// TwinCAT 3 PLC project LAMPKB
// ProgramVersion: 3.1.4023.0
// libraries:
//   LCLS General, * (SLAC)
//   lcls-twincat-motion, * (SLAC)
//   Tc2_MC2, * (Beckhoff Automation GmbH)
//   Tc2_Standard, * (Beckhoff Automation GmbH)
//   Tc2_System, * (Beckhoff Automation GmbH)
//   Tc3_Module, * (Beckhoff Automation GmbH)
// project tree:
//   / PlcTask.TcTTO
//   POUs/ FB_MotionStageStats.TcPOU, FB_PAT.TcPOU, MAIN.TcPOU
// real-time tasks:
//   TASK PlcTask: cycle T#10ms, priority 20, ADS port 350
// motion (NC):
//   TASK NC-Task 1 SAF: cycle T#2ms, priority 4, ADS port 501
//   TASK NC-Task 1 SVB: cycle T#10ms, priority 8, ADS port 511
//   AXIS MR2K4 X (id 1)
//     Dynamic: AccelerationMaximum=100, DecelerationMaximum=100, Acceleration=100, Deceleration=100, DelayTime=0.008
//     Velo: Maximum=20
//     OtherSettings: AllowMotionCmdToSlave=true
//     encoder EncType=29
//       EncPara: ScaleFactorNumerator=5e-06, Offset=-30.6825, MaxCount=#xffffffff, ReferenceSystem=1
//         Inc: RefSoftSyncMask=#x0000ffff
//     drive DrvType=24
//       DrvPara: Inverse=true
//         Analog: VeloReferenz=20, ScaleFactorActTorque=0.1
//         TimeComp: TaskDelayCycles=1
//     controller CtrType=1
//       CtrPara: PriorControlFactor=1
//         PosDiffControl: Range=0.1
//         PID: DeadBandPosition=0.001
//         Observer: BandWidth=20
//   AXIS MR2K4 Y (id 2)
//     Dynamic: AccelerationMaximum=10, DecelerationMaximum=10, Acceleration=10, Deceleration=10, Jerk=15, DelayTime=0.008
//     Velo: Maximum=1.25
//     OtherSettings: AllowMotionCmdToSlave=true
//     encoder EncType=29
//       EncPara: ScaleFactorNumerator=5e-06, Offset=-30.18, MaxCount=#xffffffff
//         Inc: RefSoftSyncMask=#x0000ffff
//     drive DrvType=24
//       DrvPara: Inverse=true
//         Analog: VeloReferenz=1.25, ScaleFactorActTorque=0.1
//         TimeComp: TaskDelayCycles=1
//     controller CtrType=1
//       CtrPara: PriorControlFactor=1
//         PosDiffControl: Range=0.1
//         Observer: BandWidth=20
//   AXIS MR2K4 rY (id 3)
//     General: UnitName=urad
//     Dynamic: AccelerationMaximum=400, DecelerationMaximum=400, Acceleration=400, Deceleration=400, Jerk=1200, DelayTime=0.008
//     Velo: Maximum=166.67
//     OtherSettings: AllowMotionCmdToSlave=true
//     encoder EncType=29
//       EncPara: ScaleFactorNumerator=0.005348, Offset=-194502.025, MaxCount=#xffffffff
//         Inc: RefSoftSyncMask=#x0000ffff
//     drive DrvType=24
//       Analog: VeloReferenz=166.67, ScaleFactorActTorque=0.1
//       TimeComp: TaskDelayCycles=1
//     controller CtrType=1
//       CtrPara: PriorControlFactor=1
//         PosDiffControl: Range=40
//         Observer: BandWidth=20
//   AXIS MR3K4 X (id 4)
//     Dynamic: AccelerationMaximum=100, DecelerationMaximum=100, Acceleration=100, Deceleration=100, DelayTime=0.008
//     Velo: Maximum=20
//     OtherSettings: AllowMotionCmdToSlave=true
//     encoder EncType=29
//       EncPara: ScaleFactorNumerator=5e-06, Offset=-31.1, MaxCount=#xffffffff
//         Inc: RefSoftSyncMask=#x0000ffff
//     drive DrvType=24
//       DrvPara: Inverse=true
//         Analog: VeloReferenz=20, ScaleFactorActTorque=0.1
//         TimeComp: TaskDelayCycles=1
//     controller CtrType=1
//       CtrPara: PriorControlFactor=1
//         PosDiffControl: Range=0.1
//         Observer: BandWidth=20
//   AXIS MR3K4 Y (id 5)
//     Dynamic: AccelerationMaximum=10, DecelerationMaximum=10, Acceleration=10, Deceleration=10, Jerk=15, DelayTime=0.008
//     Velo: Maximum=1.25
//     OtherSettings: AllowMotionCmdToSlave=true
//     encoder EncType=29
//       EncPara: ScaleFactorNumerator=5e-06, Offset=-29.68, MaxCount=#xffffffff
//         Inc: RefSoftSyncMask=#x0000ffff
//     drive DrvType=24
//       DrvPara: Inverse=true
//         Analog: VeloReferenz=1.25, ScaleFactorActTorque=0.1
//         TimeComp: TaskDelayCycles=1
//     controller CtrType=1
//       CtrPara: PriorControlFactor=1
//         PosDiffControl: Range=0.1
//         Observer: BandWidth=20
//   AXIS MR3K4 rX (id 6)
//     General: UnitName=urad
//     Dynamic: AccelerationMaximum=300, DecelerationMaximum=300, Acceleration=300, Deceleration=300, Jerk=900, DelayTime=0.008
//     Velo: Maximum=140.84
//     OtherSettings: AllowMotionCmdToSlave=true
//     encoder EncType=29
//       EncPara: ScaleFactorNumerator=0.002577, Offset=-136547, MaxCount=#xffffffff
//         Inc: RefSoftSyncMask=#x0000ffff
//     drive DrvType=24
//       Analog: VeloReferenz=140.84, ScaleFactorActTorque=0.1
//       TimeComp: TaskDelayCycles=1
//     controller CtrType=1
//       CtrPara: PriorControlFactor=1
//         PosDiffControl: Range=10
//         Observer: BandWidth=20
//   AXIS MR2K4 BEND US (id 14)
//     Dynamic: AccelerationMaximum=0.6, DecelerationMaximum=0.6, Acceleration=0.6, Deceleration=0.6, Jerk=1.2, DelayTime=0.008
//     Velo: Maximum=0.4
//     OtherSettings: AllowMotionCmdToSlave=true
//     encoder EncType=29
//       EncPara: ScaleFactorNumerator=1e-06, MaxCount=#xffffffff
//         SoftEndMinControl: Enable=true, Range=5
//         Inc: RefSoftSyncMask=#x0000ffff
//     drive DrvType=24
//       DrvPara: Inverse=true
//         Analog: VeloReferenz=0.4, ScaleFactorActTorque=0.1
//         TimeComp: TaskDelayCycles=1
//     controller CtrType=1
//       CtrPara: PriorControlFactor=1
//         PosDiffControl: Range=0.2
//         Observer: BandWidth=20
//   AXIS MR2K4 BEND DS (id 15)
//     Dynamic: AccelerationMaximum=0.6, DecelerationMaximum=0.6, Acceleration=0.6, Deceleration=0.6, Jerk=1.2, DelayTime=0.008
//     Velo: Maximum=0.1
//     OtherSettings: AllowMotionCmdToSlave=true
//     encoder EncType=29
//       EncPara: ScaleFactorNumerator=1e-06, MaxCount=#xffffffff
//         SoftEndMinControl: Enable=true, Range=5
//         Inc: RefSoftSyncMask=#x0000ffff
//     drive DrvType=24
//       DrvPara: Inverse=true
//         Analog: VeloReferenz=0.4, ScaleFactorActTorque=0.1
//         TimeComp: TaskDelayCycles=1
//     controller CtrType=1
//       CtrPara: PriorControlFactor=1
//         PosDiffControl: Range=0.2
//         Observer: BandWidth=20
//   AXIS MR3K4 BEND US (id 16)
//     Dynamic: AccelerationMaximum=0.6, DecelerationMaximum=0.6, Acceleration=0.6, Deceleration=0.6, Jerk=1.2, DelayTime=0.008
//     Velo: Maximum=0.1
//     OtherSettings: AllowMotionCmdToSlave=true
//     encoder EncType=29
//       EncPara: ScaleFactorNumerator=1e-06, MaxCount=#xffffffff
//         SoftEndMinControl: Enable=true, Range=6.25
//         Inc: RefSoftSyncMask=#x0000ffff
//     drive DrvType=24
//       DrvPara: Inverse=true
//         Analog: VeloReferenz=0.4, ScaleFactorActTorque=0.1
//         TimeComp: TaskDelayCycles=1
//     controller CtrType=1
//       CtrPara: PriorControlFactor=1
//         PosDiffControl: Range=0.2
//         Observer: BandWidth=20
//   AXIS MR3K4 BEND DS (id 17)
//     Dynamic: AccelerationMaximum=0.6, DecelerationMaximum=0.6, Acceleration=0.6, Deceleration=0.6, Jerk=1.2, DelayTime=0.008
//     Velo: Maximum=0.1
//     OtherSettings: AllowMotionCmdToSlave=true
//     encoder EncType=29
//       EncPara: ScaleFactorNumerator=1e-06, MaxCount=#xffffffff
//         SoftEndMinControl: Enable=true, Range=5.5
//         Inc: RefSoftSyncMask=#x0000ffff
//     drive DrvType=24
//       DrvPara: Inverse=true
//         Analog: VeloReferenz=0.4, ScaleFactorActTorque=0.1
//         TimeComp: TaskDelayCycles=1
//     controller CtrType=1
//       CtrPara: PriorControlFactor=1
//         PosDiffControl: Range=0.2
//         Observer: BandWidth=20
// I/O:
//   DEVICE Device 2 (EtherCAT), AmsNetId 192.168.5.67.3.1
//     Term 1 (EK1100) [EK1100 EtherCAT Coupler (2A E-Bus)]
//       Term 2 (EL5042) [EL5042 2Ch. BiSS-C Encoder]
//       Term 3 (EL5042) [EL5042 2Ch. BiSS-C Encoder]
//       Term 4 (EL5042) [EL5042 2Ch. BiSS-C Encoder]
//       MR2K4 X
//       MR2K4 Y
//       MR2K4 rY
//       MR3K4 X [EL7041-0052 1Ch. Stepper motor output stage (50V, 5A)]
//       MR3K4 Y
//       MR3K4 rX
//       Term 11 (EL9410) [EL9410 E-Bus Power Supplier  (Diagnostics)]
//       Term 12 (EL5042) [EL5042 2Ch. BiSS-C Encoder]
//       Term 13 (EL5042) [EL5042 2Ch. BiSS-C Encoder]
//       MR2K4 BEND US [EL7041 1Ch. Stepper motor output stage (50V, 5A)]
//       MR2K4 BEND DS [EL7041 1Ch. Stepper motor output stage (50V, 5A)]
//       MR3K4 BEND US
//       MR3K4 BEND DS
//       STO (EL1004) [EL1004 4Ch. Dig. Input 24V, 3ms]
//       Term 19 (EL9011) [EL9011 End Terminal]
// variable links:
//   (this object) <-> Device 2 (EtherCAT)/Term 1 (EK1100)/MR2K4 X
//     Drive/Inputs/In/nState1 @bit 3 <-> STM Status/Status/Error
//     Drive/Inputs/In/nState1 @bit 5 <-> STM Status/Status/Moving negative
//     Drive/Inputs/In/nState1 @bit 4 <-> STM Status/Status/Moving positive
//     Drive/Inputs/In/nState1 @bit 1 <-> STM Status/Status/Ready
//     Drive/Inputs/In/nState1 <-> STM Status/Status/Ready to enable
//     Drive/Inputs/In/nState1 @bit 6 <-> STM Status/Status/Torque reduced
//     Drive/Inputs/In/nState1 @bit 2 <-> STM Status/Status/Warning
//     Drive/Inputs/In/nState2 @bit 3 <-> STM Status/Status/Digital input 1
//     Drive/Inputs/In/nState2 @bit 4 <-> STM Status/Status/Digital input 2
//     Drive/Inputs/In/nState2 @bit 5 <-> STM Status/Status/Sync error
//     Drive/Inputs/In/nState2 @bit 7 <-> STM Status/Status/TxPDO Toggle
//     Drive/Inputs/In/nState4 @bit 1 <-> WcState/InputToggle
//     Drive/Inputs/In/nState4 <-> WcState/WcState
//     Drive/Outputs/Out/nCtrl1 <-> STM Control/Control/Enable
//     Drive/Outputs/Out/nCtrl1 @bit 2 <-> STM Control/Control/Reduce torque
//     Drive/Outputs/Out/nCtrl1 @bit 1 <-> STM Control/Control/Reset
//     Drive/Outputs/Out/nDataOut2[0] <-> STM Velocity/Velocity
//   (this object) <-> Device 2 (EtherCAT)/Term 1 (EK1100)/Term 2 (EL5042)
//     Enc/Inputs/In/nComState @bit 1 <-> WcState/InputToggle
//     Enc/Inputs/In/nComState <-> WcState/WcState
//     Enc/Inputs/In/nDataIn1 <-> FB Inputs Channel 1/Position
//     Enc/Inputs/In/nDataIn1 <-> FB Inputs Channel 2/Position
//     Enc/Inputs/In/nState1 @bit 12 <-> FB Inputs Channel 1/Status/Diag
//     Enc/Inputs/In/nState1 @bit 12 <-> FB Inputs Channel 2/Status/Diag
//     Enc/Inputs/In/nState1 @bit 1 <-> FB Inputs Channel 1/Status/Error
//     Enc/Inputs/In/nState1 @bit 1 <-> FB Inputs Channel 2/Status/Error
//     Enc/Inputs/In/nState1 @bit 14 <-> FB Inputs Channel 1/Status/Input cycle counter
//     Enc/Inputs/In/nState1 @bit 14 <-> FB Inputs Channel 2/Status/Input cycle counter
//     Enc/Inputs/In/nState1 @bit 2 <-> FB Inputs Channel 1/Status/Ready
//     Enc/Inputs/In/nState1 @bit 2 <-> FB Inputs Channel 2/Status/Ready
//     Enc/Inputs/In/nState1 @bit 13 <-> FB Inputs Channel 1/Status/TxPDO State
//     Enc/Inputs/In/nState1 @bit 13 <-> FB Inputs Channel 2/Status/TxPDO State
//     Enc/Inputs/In/nState1 <-> FB Inputs Channel 1/Status/Warning
//     Enc/Inputs/In/nState1 <-> FB Inputs Channel 2/Status/Warning
//   (this object) <-> Device 2 (EtherCAT)/Term 1 (EK1100)/MR2K4 Y
//     Drive/Inputs/In/nState1 @bit 3 <-> STM Status/Status/Error
//     Drive/Inputs/In/nState1 @bit 5 <-> STM Status/Status/Moving negative
//     Drive/Inputs/In/nState1 @bit 4 <-> STM Status/Status/Moving positive
//     Drive/Inputs/In/nState1 @bit 1 <-> STM Status/Status/Ready
//     Drive/Inputs/In/nState1 <-> STM Status/Status/Ready to enable
//     Drive/Inputs/In/nState1 @bit 6 <-> STM Status/Status/Torque reduced
//     Drive/Inputs/In/nState1 @bit 2 <-> STM Status/Status/Warning
//     Drive/Inputs/In/nState2 @bit 3 <-> STM Status/Status/Digital input 1
//     Drive/Inputs/In/nState2 @bit 4 <-> STM Status/Status/Digital input 2
//     Drive/Inputs/In/nState2 @bit 5 <-> STM Status/Status/Sync error
//     Drive/Inputs/In/nState2 @bit 7 <-> STM Status/Status/TxPDO Toggle
//     Drive/Inputs/In/nState4 @bit 1 <-> WcState/InputToggle
//     Drive/Inputs/In/nState4 <-> WcState/WcState
//     Drive/Outputs/Out/nCtrl1 <-> STM Control/Control/Enable
//     Drive/Outputs/Out/nCtrl1 @bit 2 <-> STM Control/Control/Reduce torque
//     Drive/Outputs/Out/nCtrl1 @bit 1 <-> STM Control/Control/Reset
//     Drive/Outputs/Out/nDataOut2[0] <-> STM Velocity/Velocity
//   (this object) <-> Device 2 (EtherCAT)/Term 1 (EK1100)/MR2K4 rY
//     Drive/Inputs/In/nState1 @bit 3 <-> STM Status/Status/Error
//     Drive/Inputs/In/nState1 @bit 5 <-> STM Status/Status/Moving negative
//     Drive/Inputs/In/nState1 @bit 4 <-> STM Status/Status/Moving positive
//     Drive/Inputs/In/nState1 @bit 1 <-> STM Status/Status/Ready
//     Drive/Inputs/In/nState1 <-> STM Status/Status/Ready to enable
//     Drive/Inputs/In/nState1 @bit 6 <-> STM Status/Status/Torque reduced
//     Drive/Inputs/In/nState1 @bit 2 <-> STM Status/Status/Warning
//     Drive/Inputs/In/nState2 @bit 3 <-> STM Status/Status/Digital input 1
//     Drive/Inputs/In/nState2 @bit 4 <-> STM Status/Status/Digital input 2
//     Drive/Inputs/In/nState2 @bit 5 <-> STM Status/Status/Sync error
//     Drive/Inputs/In/nState2 @bit 7 <-> STM Status/Status/TxPDO Toggle
//     Drive/Inputs/In/nState4 @bit 1 <-> WcState/InputToggle
//     Drive/Inputs/In/nState4 <-> WcState/WcState
//     Drive/Outputs/Out/nCtrl1 <-> STM Control/Control/Enable
//     Drive/Outputs/Out/nCtrl1 @bit 2 <-> STM Control/Control/Reduce torque
//     Drive/Outputs/Out/nCtrl1 @bit 1 <-> STM Control/Control/Reset
//     Drive/Outputs/Out/nDataOut2[0] <-> STM Velocity/Velocity
//   (this object) <-> Device 2 (EtherCAT)/Term 1 (EK1100)/Term 3 (EL5042)
//     Enc/Inputs/In/nComState @bit 1 <-> WcState/InputToggle
//     Enc/Inputs/In/nComState <-> WcState/WcState
//     Enc/Inputs/In/nDataIn1 <-> FB Inputs Channel 1/Position
//     Enc/Inputs/In/nDataIn1 <-> FB Inputs Channel 2/Position
//     Enc/Inputs/In/nState1 @bit 12 <-> FB Inputs Channel 1/Status/Diag
//     Enc/Inputs/In/nState1 @bit 12 <-> FB Inputs Channel 2/Status/Diag
//     Enc/Inputs/In/nState1 @bit 1 <-> FB Inputs Channel 1/Status/Error
//     Enc/Inputs/In/nState1 @bit 1 <-> FB Inputs Channel 2/Status/Error
//     Enc/Inputs/In/nState1 @bit 14 <-> FB Inputs Channel 1/Status/Input cycle counter
//     Enc/Inputs/In/nState1 @bit 14 <-> FB Inputs Channel 2/Status/Input cycle counter
//     Enc/Inputs/In/nState1 @bit 2 <-> FB Inputs Channel 1/Status/Ready
//     Enc/Inputs/In/nState1 @bit 2 <-> FB Inputs Channel 2/Status/Ready
//     Enc/Inputs/In/nState1 @bit 13 <-> FB Inputs Channel 1/Status/TxPDO State
//     Enc/Inputs/In/nState1 @bit 13 <-> FB Inputs Channel 2/Status/TxPDO State
//     Enc/Inputs/In/nState1 <-> FB Inputs Channel 1/Status/Warning
//     Enc/Inputs/In/nState1 <-> FB Inputs Channel 2/Status/Warning
//   (this object) <-> Device 2 (EtherCAT)/Term 1 (EK1100)/MR3K4 X
//     Drive/Inputs/In/nState1 @bit 3 <-> STM Status/Status/Error
//     Drive/Inputs/In/nState1 @bit 5 <-> STM Status/Status/Moving negative
//     Drive/Inputs/In/nState1 @bit 4 <-> STM Status/Status/Moving positive
//     Drive/Inputs/In/nState1 @bit 1 <-> STM Status/Status/Ready
//     Drive/Inputs/In/nState1 <-> STM Status/Status/Ready to enable
//     Drive/Inputs/In/nState1 @bit 6 <-> STM Status/Status/Torque reduced
//     Drive/Inputs/In/nState1 @bit 2 <-> STM Status/Status/Warning
//     Drive/Inputs/In/nState2 @bit 3 <-> STM Status/Status/Digital input 1
//     Drive/Inputs/In/nState2 @bit 4 <-> STM Status/Status/Digital input 2
//     Drive/Inputs/In/nState2 @bit 5 <-> STM Status/Status/Sync error
//     Drive/Inputs/In/nState2 @bit 7 <-> STM Status/Status/TxPDO Toggle
//     Drive/Inputs/In/nState4 @bit 1 <-> WcState/InputToggle
//     Drive/Inputs/In/nState4 <-> WcState/WcState
//     Drive/Outputs/Out/nCtrl1 <-> STM Control/Control/Enable
//     Drive/Outputs/Out/nCtrl1 @bit 2 <-> STM Control/Control/Reduce torque
//     Drive/Outputs/Out/nCtrl1 @bit 1 <-> STM Control/Control/Reset
//     Drive/Outputs/Out/nDataOut2[0] <-> STM Velocity/Velocity
//   (this object) <-> Device 2 (EtherCAT)/Term 1 (EK1100)/MR3K4 Y
//     Drive/Inputs/In/nState1 @bit 3 <-> STM Status/Status/Error
//     Drive/Inputs/In/nState1 @bit 5 <-> STM Status/Status/Moving negative
//     Drive/Inputs/In/nState1 @bit 4 <-> STM Status/Status/Moving positive
//     Drive/Inputs/In/nState1 @bit 1 <-> STM Status/Status/Ready
//     Drive/Inputs/In/nState1 <-> STM Status/Status/Ready to enable
//     Drive/Inputs/In/nState1 @bit 6 <-> STM Status/Status/Torque reduced
//     Drive/Inputs/In/nState1 @bit 2 <-> STM Status/Status/Warning
//     Drive/Inputs/In/nState2 @bit 3 <-> STM Status/Status/Digital input 1
//     Drive/Inputs/In/nState2 @bit 4 <-> STM Status/Status/Digital input 2
//     Drive/Inputs/In/nState2 @bit 5 <-> STM Status/Status/Sync error
//     Drive/Inputs/In/nState2 @bit 7 <-> STM Status/Status/TxPDO Toggle
//     Drive/Inputs/In/nState4 @bit 1 <-> WcState/InputToggle
//     Drive/Inputs/In/nState4 <-> WcState/WcState
//     Drive/Outputs/Out/nCtrl1 <-> STM Control/Control/Enable
//     Drive/Outputs/Out/nCtrl1 @bit 2 <-> STM Control/Control/Reduce torque
//     Drive/Outputs/Out/nCtrl1 @bit 1 <-> STM Control/Control/Reset
//     Drive/Outputs/Out/nDataOut2[0] <-> STM Velocity/Velocity
//   (this object) <-> Device 2 (EtherCAT)/Term 1 (EK1100)/Term 4 (EL5042)
//     Enc/Inputs/In/nComState @bit 1 <-> WcState/InputToggle
//     Enc/Inputs/In/nComState <-> WcState/WcState
//     Enc/Inputs/In/nDataIn1 <-> FB Inputs Channel 1/Position
//     Enc/Inputs/In/nDataIn1 <-> FB Inputs Channel 2/Position
//     Enc/Inputs/In/nState1 @bit 12 <-> FB Inputs Channel 1/Status/Diag
//     Enc/Inputs/In/nState1 @bit 12 <-> FB Inputs Channel 2/Status/Diag
//     Enc/Inputs/In/nState1 @bit 1 <-> FB Inputs Channel 1/Status/Error
//     Enc/Inputs/In/nState1 @bit 1 <-> FB Inputs Channel 2/Status/Error
//     Enc/Inputs/In/nState1 @bit 14 <-> FB Inputs Channel 1/Status/Input cycle counter
//     Enc/Inputs/In/nState1 @bit 14 <-> FB Inputs Channel 2/Status/Input cycle counter
//     Enc/Inputs/In/nState1 @bit 2 <-> FB Inputs Channel 1/Status/Ready
//     Enc/Inputs/In/nState1 @bit 2 <-> FB Inputs Channel 2/Status/Ready
//     Enc/Inputs/In/nState1 @bit 13 <-> FB Inputs Channel 1/Status/TxPDO State
//     Enc/Inputs/In/nState1 @bit 13 <-> FB Inputs Channel 2/Status/TxPDO State
//     Enc/Inputs/In/nState1 <-> FB Inputs Channel 1/Status/Warning
//     Enc/Inputs/In/nState1 <-> FB Inputs Channel 2/Status/Warning
//   (this object) <-> Device 2 (EtherCAT)/Term 1 (EK1100)/MR3K4 rX
//     Drive/Inputs/In/nState1 @bit 3 <-> STM Status/Status/Error
//     Drive/Inputs/In/nState1 @bit 5 <-> STM Status/Status/Moving negative
//     Drive/Inputs/In/nState1 @bit 4 <-> STM Status/Status/Moving positive
//     Drive/Inputs/In/nState1 @bit 1 <-> STM Status/Status/Ready
//     Drive/Inputs/In/nState1 <-> STM Status/Status/Ready to enable
//     Drive/Inputs/In/nState1 @bit 6 <-> STM Status/Status/Torque reduced
//     Drive/Inputs/In/nState1 @bit 2 <-> STM Status/Status/Warning
//     Drive/Inputs/In/nState2 @bit 3 <-> STM Status/Status/Digital input 1
//     Drive/Inputs/In/nState2 @bit 4 <-> STM Status/Status/Digital input 2
//     Drive/Inputs/In/nState2 @bit 5 <-> STM Status/Status/Sync error
//     Drive/Inputs/In/nState2 @bit 7 <-> STM Status/Status/TxPDO Toggle
//     Drive/Inputs/In/nState4 @bit 1 <-> WcState/InputToggle
//     Drive/Inputs/In/nState4 <-> WcState/WcState
//     Drive/Outputs/Out/nCtrl1 <-> STM Control/Control/Enable
//     Drive/Outputs/Out/nCtrl1 @bit 2 <-> STM Control/Control/Reduce torque
//     Drive/Outputs/Out/nCtrl1 @bit 1 <-> STM Control/Control/Reset
//     Drive/Outputs/Out/nDataOut2[0] <-> STM Velocity/Velocity
//   (this object) <-> Device 2 (EtherCAT)/Term 1 (EK1100)/MR2K4 BEND US
//     Drive/Inputs/In/nState1 @bit 3 <-> STM Status/Status/Error
//     Drive/Inputs/In/nState1 @bit 5 <-> STM Status/Status/Moving negative
//     Drive/Inputs/In/nState1 @bit 4 <-> STM Status/Status/Moving positive
//     Drive/Inputs/In/nState1 @bit 1 <-> STM Status/Status/Ready
//     Drive/Inputs/In/nState1 <-> STM Status/Status/Ready to enable
//     Drive/Inputs/In/nState1 @bit 6 <-> STM Status/Status/Torque reduced
//     Drive/Inputs/In/nState1 @bit 2 <-> STM Status/Status/Warning
//     Drive/Inputs/In/nState2 @bit 3 <-> STM Status/Status/Digital input 1
//     Drive/Inputs/In/nState2 @bit 4 <-> STM Status/Status/Digital input 2
//     Drive/Inputs/In/nState2 @bit 5 <-> STM Status/Status/Sync error
//     Drive/Inputs/In/nState2 @bit 7 <-> STM Status/Status/TxPDO Toggle
//     Drive/Inputs/In/nState4 @bit 1 <-> WcState/InputToggle
//     Drive/Inputs/In/nState4 <-> WcState/WcState
//     Drive/Outputs/Out/nCtrl1 <-> STM Control/Control/Enable
//     Drive/Outputs/Out/nCtrl1 @bit 2 <-> STM Control/Control/Reduce torque
//     Drive/Outputs/Out/nCtrl1 @bit 1 <-> STM Control/Control/Reset
//     Drive/Outputs/Out/nDataOut2[0] <-> STM Velocity/Velocity
//   (this object) <-> Device 2 (EtherCAT)/Term 1 (EK1100)/Term 12 (EL5042)
//     Enc/Inputs/In/nComState @bit 1 <-> WcState/InputToggle
//     Enc/Inputs/In/nComState <-> WcState/WcState
//     Enc/Inputs/In/nDataIn1 <-> FB Inputs Channel 1/Position
//     Enc/Inputs/In/nDataIn1 <-> FB Inputs Channel 2/Position
//     Enc/Inputs/In/nState1 @bit 12 <-> FB Inputs Channel 1/Status/Diag
//     Enc/Inputs/In/nState1 @bit 12 <-> FB Inputs Channel 2/Status/Diag
//     Enc/Inputs/In/nState1 @bit 1 <-> FB Inputs Channel 1/Status/Error
//     Enc/Inputs/In/nState1 @bit 1 <-> FB Inputs Channel 2/Status/Error
//     Enc/Inputs/In/nState1 @bit 14 <-> FB Inputs Channel 1/Status/Input cycle counter
//     Enc/Inputs/In/nState1 @bit 14 <-> FB Inputs Channel 2/Status/Input cycle counter
//     Enc/Inputs/In/nState1 @bit 2 <-> FB Inputs Channel 1/Status/Ready
//     Enc/Inputs/In/nState1 @bit 2 <-> FB Inputs Channel 2/Status/Ready
//     Enc/Inputs/In/nState1 @bit 13 <-> FB Inputs Channel 1/Status/TxPDO State
//     Enc/Inputs/In/nState1 @bit 13 <-> FB Inputs Channel 2/Status/TxPDO State
//     Enc/Inputs/In/nState1 <-> FB Inputs Channel 1/Status/Warning
//     Enc/Inputs/In/nState1 <-> FB Inputs Channel 2/Status/Warning
//   (this object) <-> Device 2 (EtherCAT)/Term 1 (EK1100)/MR2K4 BEND DS
//     Drive/Inputs/In/nState1 @bit 3 <-> STM Status/Status/Error
//     Drive/Inputs/In/nState1 @bit 5 <-> STM Status/Status/Moving negative
//     Drive/Inputs/In/nState1 @bit 4 <-> STM Status/Status/Moving positive
//     Drive/Inputs/In/nState1 @bit 1 <-> STM Status/Status/Ready
//     Drive/Inputs/In/nState1 <-> STM Status/Status/Ready to enable
//     Drive/Inputs/In/nState1 @bit 6 <-> STM Status/Status/Torque reduced
//     Drive/Inputs/In/nState1 @bit 2 <-> STM Status/Status/Warning
//     Drive/Inputs/In/nState2 @bit 3 <-> STM Status/Status/Digital input 1
//     Drive/Inputs/In/nState2 @bit 4 <-> STM Status/Status/Digital input 2
//     Drive/Inputs/In/nState2 @bit 5 <-> STM Status/Status/Sync error
//     Drive/Inputs/In/nState2 @bit 7 <-> STM Status/Status/TxPDO Toggle
//     Drive/Inputs/In/nState4 @bit 1 <-> WcState/InputToggle
//     Drive/Inputs/In/nState4 <-> WcState/WcState
//     Drive/Outputs/Out/nCtrl1 <-> STM Control/Control/Enable
//     Drive/Outputs/Out/nCtrl1 @bit 2 <-> STM Control/Control/Reduce torque
//     Drive/Outputs/Out/nCtrl1 @bit 1 <-> STM Control/Control/Reset
//     Drive/Outputs/Out/nDataOut2[0] <-> STM Velocity/Velocity
//   (this object) <-> Device 2 (EtherCAT)/Term 1 (EK1100)/MR3K4 BEND US
//     Drive/Inputs/In/nState1 @bit 3 <-> STM Status/Status/Error
//     Drive/Inputs/In/nState1 @bit 5 <-> STM Status/Status/Moving negative
//     Drive/Inputs/In/nState1 @bit 4 <-> STM Status/Status/Moving positive
//     Drive/Inputs/In/nState1 @bit 1 <-> STM Status/Status/Ready
//     Drive/Inputs/In/nState1 <-> STM Status/Status/Ready to enable
//     Drive/Inputs/In/nState1 @bit 6 <-> STM Status/Status/Torque reduced
//     Drive/Inputs/In/nState1 @bit 2 <-> STM Status/Status/Warning
//     Drive/Inputs/In/nState2 @bit 3 <-> STM Status/Status/Digital input 1
//     Drive/Inputs/In/nState2 @bit 4 <-> STM Status/Status/Digital input 2
//     Drive/Inputs/In/nState2 @bit 5 <-> STM Status/Status/Sync error
//     Drive/Inputs/In/nState2 @bit 7 <-> STM Status/Status/TxPDO Toggle
//     Drive/Inputs/In/nState4 @bit 1 <-> WcState/InputToggle
//     Drive/Inputs/In/nState4 <-> WcState/WcState
//     Drive/Outputs/Out/nCtrl1 <-> STM Control/Control/Enable
//     Drive/Outputs/Out/nCtrl1 @bit 2 <-> STM Control/Control/Reduce torque
//     Drive/Outputs/Out/nCtrl1 @bit 1 <-> STM Control/Control/Reset
//     Drive/Outputs/Out/nDataOut2[0] <-> STM Velocity/Velocity
//   (this object) <-> Device 2 (EtherCAT)/Term 1 (EK1100)/Term 13 (EL5042)
//     Enc/Inputs/In/nComState @bit 1 <-> WcState/InputToggle
//     Enc/Inputs/In/nComState <-> WcState/WcState
//     Enc/Inputs/In/nDataIn1 <-> FB Inputs Channel 1/Position
//     Enc/Inputs/In/nDataIn1 <-> FB Inputs Channel 2/Position
//     Enc/Inputs/In/nState1 @bit 12 <-> FB Inputs Channel 1/Status/Diag
//     Enc/Inputs/In/nState1 @bit 12 <-> FB Inputs Channel 2/Status/Diag
//     Enc/Inputs/In/nState1 @bit 1 <-> FB Inputs Channel 1/Status/Error
//     Enc/Inputs/In/nState1 @bit 1 <-> FB Inputs Channel 2/Status/Error
//     Enc/Inputs/In/nState1 @bit 14 <-> FB Inputs Channel 1/Status/Input cycle counter
//     Enc/Inputs/In/nState1 @bit 14 <-> FB Inputs Channel 2/Status/Input cycle counter
//     Enc/Inputs/In/nState1 @bit 2 <-> FB Inputs Channel 1/Status/Ready
//     Enc/Inputs/In/nState1 @bit 2 <-> FB Inputs Channel 2/Status/Ready
//     Enc/Inputs/In/nState1 @bit 13 <-> FB Inputs Channel 1/Status/TxPDO State
//     Enc/Inputs/In/nState1 @bit 13 <-> FB Inputs Channel 2/Status/TxPDO State
//     Enc/Inputs/In/nState1 <-> FB Inputs Channel 1/Status/Warning
//     Enc/Inputs/In/nState1 <-> FB Inputs Channel 2/Status/Warning
//   (this object) <-> Device 2 (EtherCAT)/Term 1 (EK1100)/MR3K4 BEND DS
//     Drive/Inputs/In/nState1 @bit 3 <-> STM Status/Status/Error
//     Drive/Inputs/In/nState1 @bit 5 <-> STM Status/Status/Moving negative
//     Drive/Inputs/In/nState1 @bit 4 <-> STM Status/Status/Moving positive
//     Drive/Inputs/In/nState1 @bit 1 <-> STM Status/Status/Ready
//     Drive/Inputs/In/nState1 <-> STM Status/Status/Ready to enable
//     Drive/Inputs/In/nState1 @bit 6 <-> STM Status/Status/Torque reduced
//     Drive/Inputs/In/nState1 @bit 2 <-> STM Status/Status/Warning
//     Drive/Inputs/In/nState2 @bit 3 <-> STM Status/Status/Digital input 1
//     Drive/Inputs/In/nState2 @bit 4 <-> STM Status/Status/Digital input 2
//     Drive/Inputs/In/nState2 @bit 5 <-> STM Status/Status/Sync error
//     Drive/Inputs/In/nState2 @bit 7 <-> STM Status/Status/TxPDO Toggle
//     Drive/Inputs/In/nState4 @bit 1 <-> WcState/InputToggle
//     Drive/Inputs/In/nState4 <-> WcState/WcState
//     Drive/Outputs/Out/nCtrl1 <-> STM Control/Control/Enable
//     Drive/Outputs/Out/nCtrl1 @bit 2 <-> STM Control/Control/Reduce torque
//     Drive/Outputs/Out/nCtrl1 @bit 1 <-> STM Control/Control/Reset
//     Drive/Outputs/Out/nDataOut2[0] <-> STM Velocity/Velocity
//   LAMPKB Instance <-> Device 2 (EtherCAT)/Term 1 (EK1100)/MR2K4 BEND DS
//     PlcTask Inputs/MAIN.M8.bLimitBackwardEnable <-> STM Status/Status/Digital input 2
//     PlcTask Inputs/MAIN.M8.bLimitForwardEnable <-> STM Status/Status/Digital input 1
//   LAMPKB Instance <-> Device 2 (EtherCAT)/Term 1 (EK1100)/MR2K4 BEND US
//     PlcTask Inputs/MAIN.M7.bLimitBackwardEnable <-> STM Status/Status/Digital input 2
//     PlcTask Inputs/MAIN.M7.bLimitForwardEnable <-> STM Status/Status/Digital input 1
//   LAMPKB Instance <-> Device 2 (EtherCAT)/Term 1 (EK1100)/MR2K4 X
//     PlcTask Inputs/MAIN.M1.bLimitBackwardEnable <-> STM Status/Status/Digital input 2
//     PlcTask Inputs/MAIN.M1.bLimitForwardEnable <-> STM Status/Status/Digital input 1
//   LAMPKB Instance <-> Device 2 (EtherCAT)/Term 1 (EK1100)/MR2K4 Y
//     PlcTask Inputs/MAIN.M2.bLimitBackwardEnable <-> STM Status/Status/Digital input 2
//     PlcTask Inputs/MAIN.M2.bLimitForwardEnable <-> STM Status/Status/Digital input 1
//   LAMPKB Instance <-> Device 2 (EtherCAT)/Term 1 (EK1100)/MR2K4 rY
//     PlcTask Inputs/MAIN.M3.bLimitBackwardEnable <-> STM Status/Status/Digital input 2
//     PlcTask Inputs/MAIN.M3.bLimitForwardEnable <-> STM Status/Status/Digital input 1
//   LAMPKB Instance <-> Device 2 (EtherCAT)/Term 1 (EK1100)/MR3K4 BEND DS
//     PlcTask Inputs/MAIN.M10.bLimitBackwardEnable <-> STM Status/Status/Digital input 2
//     PlcTask Inputs/MAIN.M10.bLimitForwardEnable <-> STM Status/Status/Digital input 1
//   LAMPKB Instance <-> Device 2 (EtherCAT)/Term 1 (EK1100)/MR3K4 BEND US
//     PlcTask Inputs/MAIN.M9.bLimitBackwardEnable <-> STM Status/Status/Digital input 2
//     PlcTask Inputs/MAIN.M9.bLimitForwardEnable <-> STM Status/Status/Digital input 1
//   LAMPKB Instance <-> Device 2 (EtherCAT)/Term 1 (EK1100)/MR3K4 X
//     PlcTask Inputs/MAIN.M4.bLimitBackwardEnable <-> STM Status/Status/Digital input 2
//     PlcTask Inputs/MAIN.M4.bLimitForwardEnable <-> STM Status/Status/Digital input 1
//   LAMPKB Instance <-> Device 2 (EtherCAT)/Term 1 (EK1100)/MR3K4 Y
//     PlcTask Inputs/MAIN.M5.bLimitBackwardEnable <-> STM Status/Status/Digital input 2
//     PlcTask Inputs/MAIN.M5.bLimitForwardEnable <-> STM Status/Status/Digital input 1
//   LAMPKB Instance <-> Device 2 (EtherCAT)/Term 1 (EK1100)/MR3K4 rX
//     PlcTask Inputs/MAIN.M6.bLimitBackwardEnable <-> STM Status/Status/Digital input 2
//     PlcTask Inputs/MAIN.M6.bLimitForwardEnable <-> STM Status/Status/Digital input 1
//   LAMPKB Instance <-> Device 2 (EtherCAT)/Term 1 (EK1100)/STO (EL1004)
//     PlcTask Inputs/MAIN.bSTOEnable1 <-> Channel 1/Input
//     PlcTask Inputs/MAIN.bSTOEnable2 <-> Channel 2/Input
//   LAMPKB Instance <-> NC-Task 1 SAF/Axes/MR2K4 BEND DS
//     PlcTask Inputs/MAIN.M8.Axis.NcToPlc <-> Outputs/ToPlc
//     PlcTask Outputs/MAIN.M8.Axis.PlcToNc <-> Inputs/FromPlc
//   LAMPKB Instance <-> NC-Task 1 SAF/Axes/MR2K4 BEND US
//     PlcTask Inputs/MAIN.M7.Axis.NcToPlc <-> Outputs/ToPlc
//     PlcTask Outputs/MAIN.M7.Axis.PlcToNc <-> Inputs/FromPlc
//   LAMPKB Instance <-> NC-Task 1 SAF/Axes/MR2K4 X
//     PlcTask Inputs/MAIN.M1.Axis.NcToPlc <-> Outputs/ToPlc
//     PlcTask Outputs/MAIN.M1.Axis.PlcToNc <-> Inputs/FromPlc
//   LAMPKB Instance <-> NC-Task 1 SAF/Axes/MR2K4 Y
//     PlcTask Inputs/MAIN.M2.Axis.NcToPlc <-> Outputs/ToPlc
//     PlcTask Outputs/MAIN.M2.Axis.PlcToNc <-> Inputs/FromPlc
//   LAMPKB Instance <-> NC-Task 1 SAF/Axes/MR2K4 rY
//     PlcTask Inputs/MAIN.M3.Axis.NcToPlc <-> Outputs/ToPlc
//     PlcTask Outputs/MAIN.M3.Axis.PlcToNc <-> Inputs/FromPlc
//   LAMPKB Instance <-> NC-Task 1 SAF/Axes/MR3K4 BEND DS
//     PlcTask Inputs/MAIN.M10.Axis.NcToPlc <-> Outputs/ToPlc
//     PlcTask Outputs/MAIN.M10.Axis.PlcToNc <-> Inputs/FromPlc
//   LAMPKB Instance <-> NC-Task 1 SAF/Axes/MR3K4 BEND US
//     PlcTask Inputs/MAIN.M9.Axis.NcToPlc <-> Outputs/ToPlc
//     PlcTask Outputs/MAIN.M9.Axis.PlcToNc <-> Inputs/FromPlc
//   LAMPKB Instance <-> NC-Task 1 SAF/Axes/MR3K4 X
//     PlcTask Inputs/MAIN.M4.Axis.NcToPlc <-> Outputs/ToPlc
//     PlcTask Outputs/MAIN.M4.Axis.PlcToNc <-> Inputs/FromPlc
//   LAMPKB Instance <-> NC-Task 1 SAF/Axes/MR3K4 Y
//     PlcTask Inputs/MAIN.M5.Axis.NcToPlc <-> Outputs/ToPlc
//     PlcTask Outputs/MAIN.M5.Axis.PlcToNc <-> Inputs/FromPlc
//   LAMPKB Instance <-> NC-Task 1 SAF/Axes/MR3K4 rX
//     PlcTask Inputs/MAIN.M6.Axis.NcToPlc <-> Outputs/ToPlc
//     PlcTask Outputs/MAIN.M6.Axis.PlcToNc <-> Inputs/FromPlc

CONFIGURATION LAMPKB
    RESOURCE PLC ON TwinCAT3
        TASK PlcTask(INTERVAL := T#10ms, PRIORITY := 20);
        PROGRAM MAIN WITH PlcTask : MAIN;
    END_RESOURCE
END_CONFIGURATION

// ---- POUs/MAIN.TcPOU
PROGRAM MAIN
VAR
	//MR2K4 X
	{attribute 'TcLinkTo' := '.bLimitForwardEnable:=TIIB[MR2K4 X]^STM Status^Status^Digital input 1;
                              .bLimitBackwardEnable:=TIIB[MR2K4 X]^STM Status^Status^Digital input 2'}
	{attribute 'pytmc' := '
		pv: MR2K4:MMS:X
	'}
	M1 : DUT_MotionStage := (nEnableMode:=ENUM_StageEnableMode.ALWAYS);
	fbMotionStageM1 : FB_MotionStage;
	//MR2K4 Y
	{attribute 'TcLinkTo' := '.bLimitForwardEnable:=TIIB[MR2K4 Y]^STM Status^Status^Digital input 1;
                              .bLimitBackwardEnable:=TIIB[MR2K4 Y]^STM Status^Status^Digital input 2'}
	{attribute 'pytmc' := '
		pv: MR2K4:MMS:Y
	'}
	M2 : DUT_MotionStage := (nEnableMode:=ENUM_StageEnableMode.ALWAYS);
	fbMotionStageM2 : FB_MotionStage;
	//MR2K4 rY
	{attribute 'TcLinkTo' := '.bLimitForwardEnable:=TIIB[MR2K4 rY]^STM Status^Status^Digital input 1;
                              .bLimitBackwardEnable:=TIIB[MR2K4 rY]^STM Status^Status^Digital input 2'}
	{attribute 'pytmc' := '
		pv: MR2K4:MMS:rY
	'}
	M3 : DUT_MotionStage := (nEnableMode:=ENUM_StageEnableMode.ALWAYS);
	fbMotionStageM3 : FB_MotionStage;
	//MR3K4 X
	{attribute 'TcLinkTo' := '.bLimitForwardEnable:=TIIB[MR3K4 X]^STM Status^Status^Digital input 1;
                              .bLimitBackwardEnable:=TIIB[MR3K4 X]^STM Status^Status^Digital input 2'}
	{attribute 'pytmc' := '
		pv: MR3K4:MMS:X
	'}
	M4 : DUT_MotionStage := (nEnableMode:=ENUM_StageEnableMode.ALWAYS);
	fbMotionStageM4 : FB_MotionStage;
	//MR3K4 Y
	{attribute 'TcLinkTo' := '.bLimitForwardEnable:=TIIB[MR3K4 Y]^STM Status^Status^Digital input 1;
                              .bLimitBackwardEnable:=TIIB[MR3K4 Y]^STM Status^Status^Digital input 2'}
	{attribute 'pytmc' := '
		pv: MR3K4:MMS:Y
	'}
	M5 : DUT_MotionStage := (nEnableMode:=ENUM_StageEnableMode.ALWAYS);
	fbMotionStageM5 : FB_MotionStage;
	//MR3K4 rX
	{attribute 'TcLinkTo' := '.bLimitForwardEnable:=TIIB[MR3K4 rX]^STM Status^Status^Digital input 1;
                              .bLimitBackwardEnable:=TIIB[MR3K4 rX]^STM Status^Status^Digital input 2'}
	{attribute 'pytmc' := '
		pv: MR3K4:MMS:rX
	'}
	M6 : DUT_MotionStage := (nEnableMode:=ENUM_StageEnableMode.ALWAYS);
	fbMotionStageM6 : FB_MotionStage;
	//MR2K4 US BEND
	{attribute 'TcLinkTo' := '.bLimitForwardEnable:=TIIB[MR2K4 BEND US]^STM Status^Status^Digital input 1;
							  .bLimitBackwardEnable:=TIIB[MR2K4 BEND US]^STM Status^Status^Digital input 2'}
	{attribute 'pytmc' := '
		pv: MR2K4:BEND:MMS:US
	'}
	M7 : DUT_MotionStage := (nEnableMode:=ENUM_StageEnableMode.ALWAYS);
	fbMotionStageM7 : FB_MotionStage;
	//MR2K4 DS BEND
	{attribute 'TcLinkTo' := '.bLimitForwardEnable:=TIIB[MR2K4 BEND DS]^STM Status^Status^Digital input 1;
                              .bLimitBackwardEnable:=TIIB[MR2K4 BEND DS]^STM Status^Status^Digital input 2'}
	{attribute 'pytmc' := '
		pv: MR2K4:BEND:MMS:DS
	'}
	M8 : DUT_MotionStage := (nEnableMode:=ENUM_StageEnableMode.ALWAYS);
	fbMotionStageM8 : FB_MotionStage;
	//MR3K4 US BEND
	{attribute 'TcLinkTo' := '.bLimitForwardEnable:=TIIB[MR3K4 BEND US]^STM Status^Status^Digital input 1;
                              .bLimitBackwardEnable:=TIIB[MR3K4 BEND US]^STM Status^Status^Digital input 2'}
	{attribute 'pytmc' := '
		pv: MR3K4:BEND:MMS:US
	'}
	M9 : DUT_MotionStage := (nEnableMode:=ENUM_StageEnableMode.ALWAYS);
	fbMotionStageM9 : FB_MotionStage;
	//MR3K4 DS BEND
	{attribute 'TcLinkTo' := '.bLimitForwardEnable:=TIIB[MR3K4 BEND DS]^STM Status^Status^Digital input 1;
                              .bLimitBackwardEnable:=TIIB[MR3K4 BEND DS]^STM Status^Status^Digital input 2'}
	{attribute 'pytmc' := '
		pv: MR3K4:BEND:MMS:DS
	'}
	M10 : DUT_MotionStage := (nEnableMode:=ENUM_StageEnableMode.ALWAYS);
	fbMotionStageM10 : FB_MotionStage;
	
	//MR2K4 stats
	fbM1Stats : FB_MotionStageStats;
	fbM2Stats : FB_MotionStageStats;
	fbM3Stats : FB_MotionStageStats;
	//MR3K4 stats
	fbM4Stats : FB_MotionStageStats;
	fbM5Stats : FB_MotionStageStats;
	fbM6Stats : FB_MotionStageStats;
	//MR2K4 BEND stats
	fbM7Stats : FB_MotionStageStats;
	fbM8Stats : FB_MotionStageStats;
	//MR3K4 BEND stats
	fbM9Stats : FB_MotionStageStats;	
	fbM10Stats : FB_MotionStageStats;
	
	//Emergency Stop
	bSTOEnable1 AT %I* : BOOL;
	bSTOEnable2 AT %I* : BOOL;
	
END_VAR

//MR2K4
M1.bHardwareEnable := bSTOEnable1 AND bSTOEnable2;
M2.bHardwareEnable := bSTOEnable1 AND bSTOEnable2;
M3.bHardwareEnable := bSTOEnable1 AND bSTOEnable2;
//MR3K4
M4.bHardwareEnable := bSTOEnable1 AND bSTOEnable2;
M5.bHardwareEnable := bSTOEnable1 AND bSTOEnable2;
M6.bHardwareEnable := bSTOEnable1 AND bSTOEnable2;
//MR2K4 BEND
M7.bHardwareEnable := bSTOEnable1 AND bSTOEnable2;
M8.bHardwareEnable := bSTOEnable1 AND bSTOEnable2;
//MR3K4 BEND
M9.bHardwareEnable := bSTOEnable1 AND bSTOEnable2;
M10.bHardwareEnable := bSTOEnable1 AND bSTOEnable2;

//MR2K4
fbMotionStageM1(stMotionStage:=M1);
fbMotionStageM2(stMotionStage:=M2);
fbMotionStageM3(stMotionStage:=M3);
//MR3K4
fbMotionStageM4(stMotionStage:=M4);
fbMotionStageM5(stMotionStage:=M5);
fbMotionStageM6(stMotionStage:=M6);
//MR2K4 BEND
fbMotionStageM7(stMotionStage:=M7);
fbMotionStageM8(stMotionStage:=M8);
//MR3K4 BEND
fbMotionStageM9(stMotionStage:=M9);
fbMotionStageM10(stMotionStage:=M10);

//MR2K4
fbM1Stats(Axis:=M1);
fbM2Stats(Axis:=M2);
fbM3Stats(Axis:=M3);
//MR3K4
fbM4Stats(Axis:=M4);
fbM5Stats(Axis:=M5);
fbM6Stats(Axis:=M6);
//MR2K4 BEND
fbM7Stats(Axis:=M7);
fbM8Stats(Axis:=M8);
//MR3K4 BEND
fbM9Stats(Axis:=M9);
fbM10Stats(Axis:=M10);

END_PROGRAM

// ---- POUs/FB_MotionStageStats.TcPOU
FUNCTION_BLOCK FB_MotionStageStats EXTENDS FB_BasicStats
VAR_INPUT
	Axis : DUT_MotionStage;
END_VAR
VAR_OUTPUT
END_VAR
VAR
	aActPos : ARRAY [0..ARRAY_SIZE] OF LREAL;
	idx: UINT;
END_VAR
VAR CONSTANT
	ARRAY_SIZE : UINT := 500;
END_VAR


aActPos[idx] := Axis.Axis.NcToPlc.ActPos;

idx := (idx + 1) MOD ARRAY_SIZE;

SUPER^(aSignal:=aActPos, bAlwaysCalc:=NOT bReset);

END_FUNCTION_BLOCK

// ---- POUs/FB_PAT.TcPOU
FUNCTION_BLOCK FB_PAT
VAR_INPUT
	Velocity : LREAL;
END_VAR
VAR_OUTPUT
	FwLimPos : LREAL; // Positive limit position
	BwLimPos : LREAL; // 
END_VAR
VAR_IN_OUT
	Stage : DUT_MotionStage;
END_VAR
VAR
	fbMicroStepCount : FB_MicroStepCountTest;
	
	fbMove: MC_Jog;
	tFwLim: F_TRIG;
	tBwLim: F_TRIG;
	Dir: INT;
END_VAR



// Relative move until limit, reverse and repeat, record positions, do math and spit out travel range

tFwLim(CLK:=Stage.bLimitForwardEnable);
tBwLim(CLK:=Stage.bLimitBackwardEnable);

WHILE Stage.bLimitBackwardEnable AND Stage.bLimitForwardEnable DO
	IF tFwLim.Q OR tBwLim.Q THEN
		IF (Dir = 1 AND tBwLim.Q) OR (Dir = -1 AND tFwLim.Q) THEN
			// Error, limits backwards
			EXIT;
		END_IF
		
		IF tFwLim.Q THEN
			FwLimPos := Stage.Axis.NcToPlc.ActPos;
		ELSIF tBwLim.Q THEN
			BwLimPos := Stage.Axis.NcToPlc.ActPos;
		END_IF
		
		
	END_IF
	
	
	
END_WHILE

// Discover minimum step size in one direction

// Attempt minimum step size in alternating direction

fbMove(Axis:=Stage.Axis, Velocity:=Velocity, Mode:=E_JogMode.MC_JOGMODE_CONTINOUS);

END_FUNCTION_BLOCK
